(*
SPDX-FileCopyrightText: © 2026 Oleksandr Tiutyk <trofimich@gmail.com>
SPDX-License-Identifier: MIT
License: https://opensource.org/license/mit
*)

(*!
<summary>Provides FIFO head inspection, indexed access and membership queries.</summary>
<description>
Returned descriptors and payload are borrowed, not clones. Do not modify descriptor metadata or release
payload through this view, even when IsMemoryOwner is TRUE. Keep the source and borrowed storage alive;
mutation or destruction can invalidate the view. ContainsGeneric currently defaults to releasing an owned
query.
</description>
*)

INTERFACE IReadOnlyQueue EXTENDS ICollection

(*!
<summary>Searches for a value using default generic equality.</summary>
<description>
Borrows the ANY argument during a linear search without cloning or releasing it. isObject = TRUE means a live
Object FB instance, not a pointer or interface variable. Equality exceptions propagate; callbacks that mutate
the collection can invalidate traversal.
</description>
*)
METHOD Contains : BOOL
VAR_INPUT
	value : ANY;
	isObject : BOOL := FALSE;
END_VAR
END_METHOD

(*!
<summary>Searches for an equal generic value and optionally releases the query.</summary>
<description>
Uses GENERIC_VALUE.Equals in a linear search. releaseValue defaults to TRUE: after a completed search, Release
is called on the local query copy, including on a miss. Caller-side aliases are not reset. The query must not
own storage retained by the collection. Requested release is attempted after both successful lookup and lookup
failure. Before cleanup, the original framework exception is retained and a borrowed static system exception
is cloned to preserve its code, catch point and timestamps across cleanup callbacks. The captured exception is
then propagated through ExceptionManager.Throw in the current cyclic task; native errors use the framework
SystemException representation. If capturing the system exception fails with terminal OOM, query cleanup is
still attempted and terminal OOM takes precedence. Terminal allocation state is never cleared. Release is best
effort and does not prove successful deallocation. Cleanup callbacks must not reenter collection mutation.
</description>
*)
METHOD ContainsGeneric : BOOL
VAR_INPUT
	value : TOF_Core.GENERIC_VALUE;
	releaseValue : BOOL := TRUE;
END_VAR
END_METHOD

(*!
<summary>Borrows the descriptor at a zero-based queue position.</summary>
<description>
Position zero is the head. An out-of-range index raises an exception. Returned descriptors and payload are
borrowed, not clones. Do not modify descriptor metadata or release payload through this view, even when
IsMemoryOwner is TRUE. Keep the source and borrowed storage alive; mutation or destruction can invalidate the
view.
</description>
*)
METHOD GetByIndex : REFERENCE TO TOF_Core.GENERIC_VALUE
VAR_INPUT
	index : TOF_Core.DINT_INDEX;
END_VAR
END_METHOD

(*!
<summary>Borrows the FIFO head without removing it.</summary>
<description>
An empty queue raises CollectionEmptyException. Returned descriptors and payload are borrowed, not clones. Do
not modify descriptor metadata or release payload through this view, even when IsMemoryOwner is TRUE. Keep the
source and borrowed storage alive; mutation or destruction can invalidate the view.
</description>
*)
METHOD Peek : REFERENCE TO TOF_Core.GENERIC_VALUE
END_METHOD

END_INTERFACE

(* stored: Version 1.1.0.1
   Itf IReadOnlyQueue: Id {495921cf-52ef-4089-a0ee-1dd33e33b46a}
   Method Contains: Id {568f9017-3ac6-4241-b298-87736f73468b}
   Method ContainsGeneric: Id {b784ff88-d555-4ac8-b89e-846abd0b6644}
   Method GetByIndex: Id {28e92834-617f-4705-a682-aaa3b18e78f7}
   Method Peek: Id {3b3b0174-6662-49b9-a00b-6555d4a4415a} *)
